// Mitsubishi GX Works2 project: k09   PLC: Q02/Q02H

PROGRAM MAIN
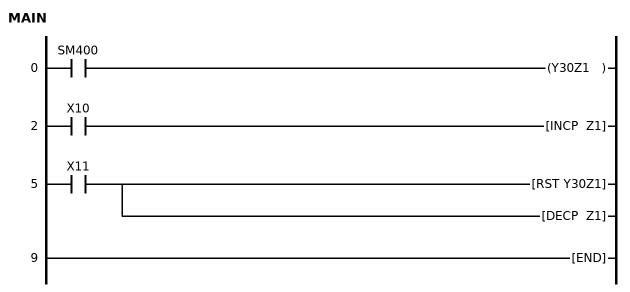
0     LD      SM400
      OUT     Y30Z1
2     LD      X10
      INCP    Z1
5     LD      X11
      RST     Y30Z1
      DECP    Z1
9     END
END_PROGRAM
